(* CoDeSys 2.3.9.47 project: lab_4_lib.pro *)
(* Libraries: C:\Users\Raphael\Documents\HSLU\05_HS_16\ATS\sharedFolder\Projects\Lab_4\lib_lab_4.lib*17.11.16 20:23:40, STANDARD.LIB 5.6.98 11:03:02 *)

(* Task configuration *)
TASK Standard (PRIORITY := 0, INTERVAL := T#1ms);
	MAIN
END_TASK

(* POU MAIN, ST *)
PROGRAM MAIN
VAR
(* Variables part A *)
(**)
INT25	: 	Integrator; 
INT50	: 	Integrator; 
INT75	: 	Integrator;
(**)
LP010	:	LowpassFilter;
LP001	:	LowpassFilter;
LP100	:	LowpassFilter;
(**)
LP010SQ	:	LowpassFilter;
LP001SQ	:	LowpassFilter;
LP100SQ	:	LowpassFilter;
(**)
SOL010	:	SecondOrderLag;
SOL001	:	SecondOrderLag;
SOL100	:	SecondOrderLag;
wr		:	REAL;

END_VAR
t_cycle := 0.001;
(* Part A *)
(*Integrators*)
INT25(); INT25.e_k := PWMSignal(t_global,25,5);
INT50(); INT50.e_k := PWMSignal(t_global,50,5);
INT75(); INT75.e_k := PWMSignal(t_global,75,5);

LP010(); LP010.tau := 0.1; LP010.x_k := SinusFunction(t_global,10);
LP001(); LP001.tau := 0.1; LP001.x_k := SinusFunction(t_global,1);
LP100(); LP100.tau := 0.1; LP100.x_k := SinusFunction(t_global,100);
(**)

LP010SQ(); LP010SQ.tau := 0.1; LP010SQ.x_k := PWMSignal(t_global,50,(2*3.14)/10);
LP001SQ(); LP001SQ.tau := 0.1; LP001SQ.x_k := PWMSignal(t_global,50,(2*3.14)/1);
LP100SQ(); LP100SQ.tau := 0.1; LP100SQ.x_k := PWMSignal(t_global,50,(2*3.14)/100);

wr := 10*SQRT(1-2*EXPT(0.2,2));
SOL010(); SOL010.w0 := 10; SOL010.d := 0.2;
SOL010.x_k := SinusFunction(t_global,wr/10);

SOL001(); SOL001.w0 := 10; SOL001.d := 0.2;
SOL001.x_k := SinusFunction(t_global,wr/1);


SOL100(); SOL100.w0 := 10; SOL100.d := 0.2;
SOL100.x_k := SinusFunction(t_global,wr*10);


(*Increment Time*)
t_global := t_global + t_cycle;
END_PROGRAM
